// Mitsubishi GX Works2 project: e05   PLC: Q02/Q02H

PROGRAM MAIN
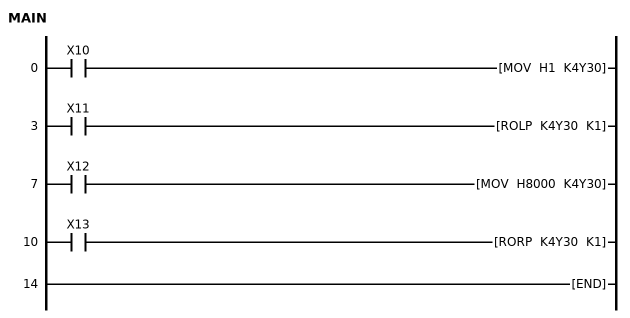
0     LD      X10
      MOV     H1 K4Y30
3     LD      X11
      ROLP    K4Y30 K1
7     LD      X12
      MOV     H8000 K4Y30
10    LD      X13
      RORP    K4Y30 K1
14    END
END_PROGRAM
